INTERFACE I_GCode

PROPERTY P_Return : REFERENCE to ST_CommandReturn
GET
END_GET
END_PROPERTY

METHOD StartMovement
VAR_INPUT
	sFilePath	: STRING;
END_VAR
END_METHOD

END_INTERFACE

(* stored: Version 1.1.0.1
   Itf I_GCode: Id {d5a3f934-6338-4630-8d61-d9069679b4c0}
   Property P_Return: Id {178a2d40-d450-4d2a-876f-2a1956770d9b}
   Get Get: Id {ddfd7fe4-419d-4342-a773-c7e770e400bd}
   Method StartMovement: Id {18ca137f-abc1-4d79-84fb-19ec6961689a} *)
